(* Logix 5000 project; controller DUNEW2PLC1 vendor 1 type 14 code 221 rev 33.11; software revision 33.00; part 4 of 4 *)
(* tags used below, declared in another part *)
   ALL_EOT_GOOD : BOOL;
   HomeTrigger : BOOL;
   INIT_DONE : BOOL;
   MORE_STATS_S : BOOL[32];
   MOVE_TYPE : INT;   // 0 = No Move 1 = XY JOG 2 = XY Plane Move 3 = Z JOG 4 = Z Axis Move 5 = Toggle Latch Actuator 6 = Home the Latch Actuator
   NEXTSTATE : DINT;
   resetPB_S : BOOL;
   Safety_System_Healthy : BOOL;
   Safety_Tripped_S : BOOL;
   STATE : DINT;   // CURRENT State Machine State
   X_axis : AXIS_CIP_DRIVE;
   X_Axis_SFX : SAFETY_FEEDBACK_INTERFACE;
   X_Axis_SLS : SAFELY_LIMITED_SPEED;
   Y_axis : AXIS_CIP_DRIVE;
   Z_axis : AXIS_CIP_DRIVE;

PROGRAM Ready_State_1   (* main routine Ready *)
VAR
   OutBit : BOOL[32];
   SetBit : BOOL[32];
   STATE1_IND : BOOL := 1; {access Read Only}
END_VAR

ROUTINE Ready   (* ladder *)
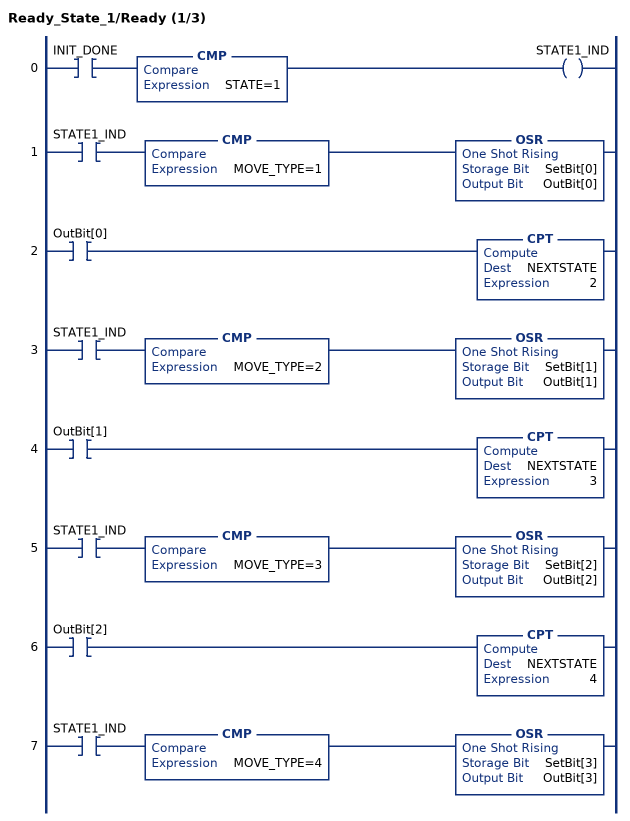
   0: XIC(INIT_DONE)CMP(STATE=1)OTE(STATE1_IND);
   1: XIC(STATE1_IND)CMP(MOVE_TYPE=1)OSR(SetBit[0],OutBit[0]);
   2: XIC(OutBit[0])CPT(NEXTSTATE,2);
   3: XIC(STATE1_IND)CMP(MOVE_TYPE=2)OSR(SetBit[1],OutBit[1]);
   4: XIC(OutBit[1])CPT(NEXTSTATE,3);
   5: XIC(STATE1_IND)CMP(MOVE_TYPE=3)OSR(SetBit[2],OutBit[2]);
   6: XIC(OutBit[2])CPT(NEXTSTATE,4);
   7: XIC(STATE1_IND)CMP(MOVE_TYPE=4)OSR(SetBit[3],OutBit[3]);
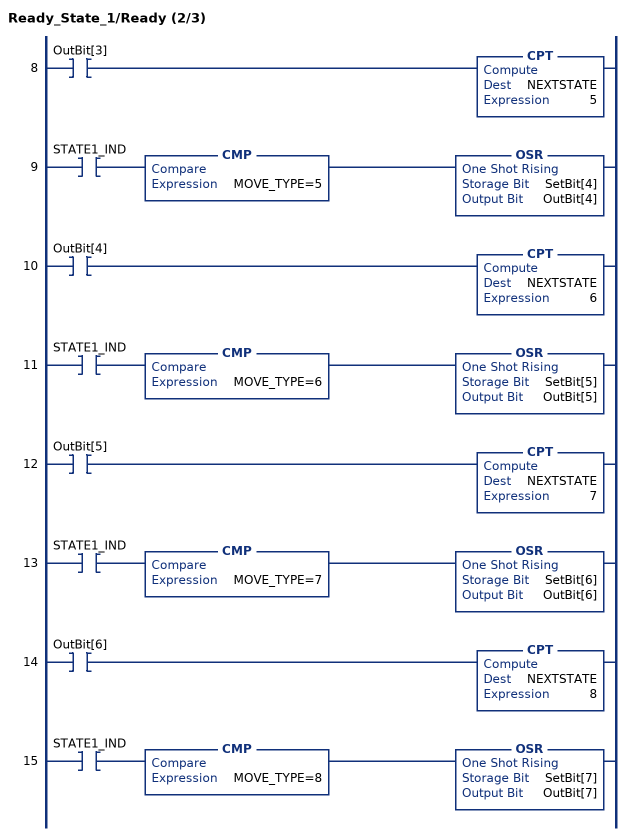
   8: XIC(OutBit[3])CPT(NEXTSTATE,5);
   9: XIC(STATE1_IND)CMP(MOVE_TYPE=5)OSR(SetBit[4],OutBit[4]);
   10: XIC(OutBit[4])CPT(NEXTSTATE,6);
   11: XIC(STATE1_IND)CMP(MOVE_TYPE=6)OSR(SetBit[5],OutBit[5]);
   12: XIC(OutBit[5])CPT(NEXTSTATE,7);
   13: XIC(STATE1_IND)CMP(MOVE_TYPE=7)OSR(SetBit[6],OutBit[6]);
   14: XIC(OutBit[6])CPT(NEXTSTATE,8);
   15: XIC(STATE1_IND)CMP(MOVE_TYPE=8)OSR(SetBit[7],OutBit[7]);
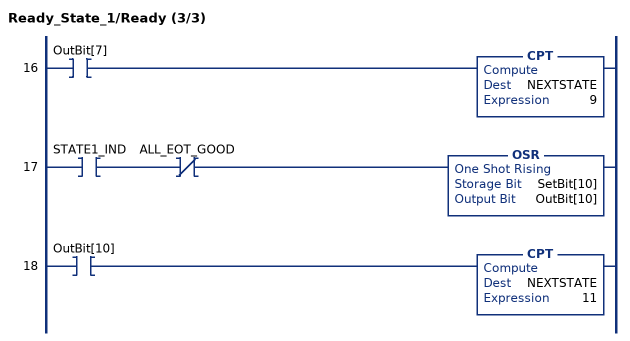
   16: XIC(OutBit[7])CPT(NEXTSTATE,9);
   17 (stored rung type 4): XIC(STATE1_IND)XIO(ALL_EOT_GOOD)OSR(SetBit[10],OutBit[10]);
   18 (stored rung type 4): XIC(OutBit[10])CPT(NEXTSTATE,11);
END_ROUTINE
END_PROGRAM

PROGRAM Safety   (* main routine Safety, safety *)
VAR
   e : BOOL;
   Machine_Reduced_Speed : BOOL;
END_VAR

ROUTINE Safety   (* ladder *)
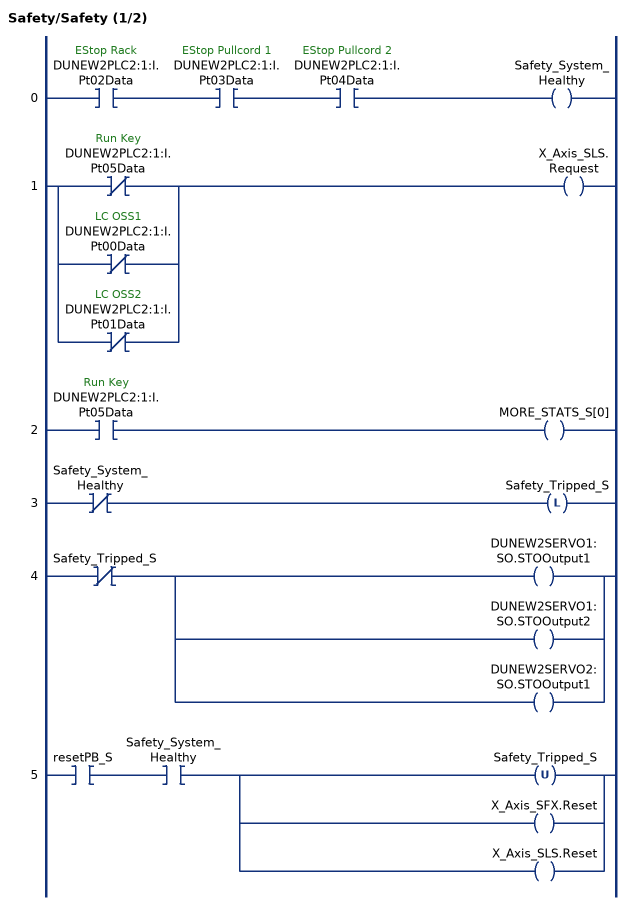
   0: XIC(DUNEW2PLC2:1:I.Pt02Data)XIC(DUNEW2PLC2:1:I.Pt03Data)XIC(DUNEW2PLC2:1:I.Pt04Data)OTE(Safety_System_Healthy);
   1: [XIO(DUNEW2PLC2:1:I.Pt05Data) ,XIO(DUNEW2PLC2:1:I.Pt00Data) ,XIO(DUNEW2PLC2:1:I.Pt01Data) ]OTE(X_Axis_SLS.Request);
   2: XIC(DUNEW2PLC2:1:I.Pt05Data)OTE(MORE_STATS_S[0]);
   3: XIO(Safety_System_Healthy)OTL(Safety_Tripped_S);
   4: XIO(Safety_Tripped_S)[[OTE(DUNEW2SERVO1:SO.STOOutput1) ,OTE(DUNEW2SERVO1:SO.STOOutput2) ] ,OTE(DUNEW2SERVO2:SO.STOOutput1) ];
   5: XIC(resetPB_S)XIC(Safety_System_Healthy)[OTU(Safety_Tripped_S) ,[OTE(X_Axis_SFX.Reset) ,OTE(X_Axis_SLS.Reset) ] ];
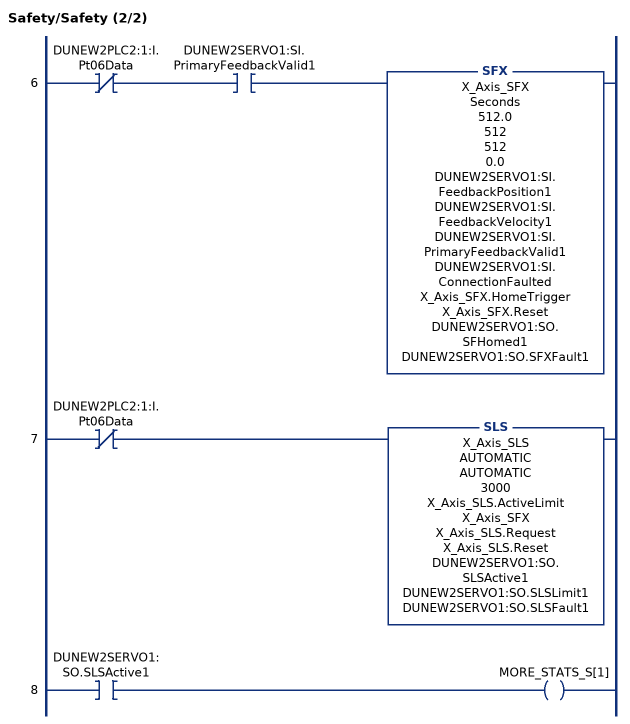
   6: XIO(DUNEW2PLC2:1:I.Pt06Data)XIC(DUNEW2SERVO1:SI.PrimaryFeedbackValid1)SFX(X_Axis_SFX,Seconds,512.0,512,512,0.0,DUNEW2SERVO1:SI.FeedbackPosition1,DUNEW2SERVO1:SI.FeedbackVelocity1,DUNEW2SERVO1:SI.PrimaryFeedbackValid1,DUNEW2SERVO1:SI.ConnectionFaulted,X_Axis_SFX.HomeTrigger,X_Axis_SFX.Reset,DUNEW2SERVO1:SO.SFHomed1,DUNEW2SERVO1:SO.SFXFault1);
   7: XIO(DUNEW2PLC2:1:I.Pt06Data)SLS(X_Axis_SLS,AUTOMATIC,AUTOMATIC,3000,X_Axis_SLS.ActiveLimit,X_Axis_SFX,X_Axis_SLS.Request,X_Axis_SLS.Reset,DUNEW2SERVO1:SO.SLSActive1,DUNEW2SERVO1:SO.SLSLimit1,DUNEW2SERVO1:SO.SLSFault1);
   8: XIC(DUNEW2SERVO1:SO.SLSActive1)OTE(MORE_STATS_S[1]);
END_ROUTINE
END_PROGRAM

PROGRAM UnServo_9   (* main routine UnServo_All *)
VAR
   oneshotob : BOOL[32]; {access Read Only}
   oneshotsb : BOOL[32]; {access Read Only}
   STATE9_IND : BOOL; {access Read Only}
   X_AXIS_STAT : MOTION_INSTRUCTION[32] := ([0].FLAGS := 33554432, [1].FLAGS := 33554432, [2].FLAGS := 536870912, [2].DN := 1, [2].STATE := 1); {access Read Only}
   Y_AXIS_STAT : MOTION_INSTRUCTION[32] := ([0].FLAGS := 33554432, [1].FLAGS := 33554432, [2].FLAGS := 536870912, [2].DN := 1, [2].STATE := 1); {access Read Only}
   Z_AXIS_STAT : MOTION_INSTRUCTION[32] := ([0].FLAGS := 33554432, [1].FLAGS := 33554432, [2].FLAGS := 536870912, [2].DN := 1, [2].STATE := 1); {access Read Only}
END_VAR

ROUTINE UnServo_All   (* ladder *)
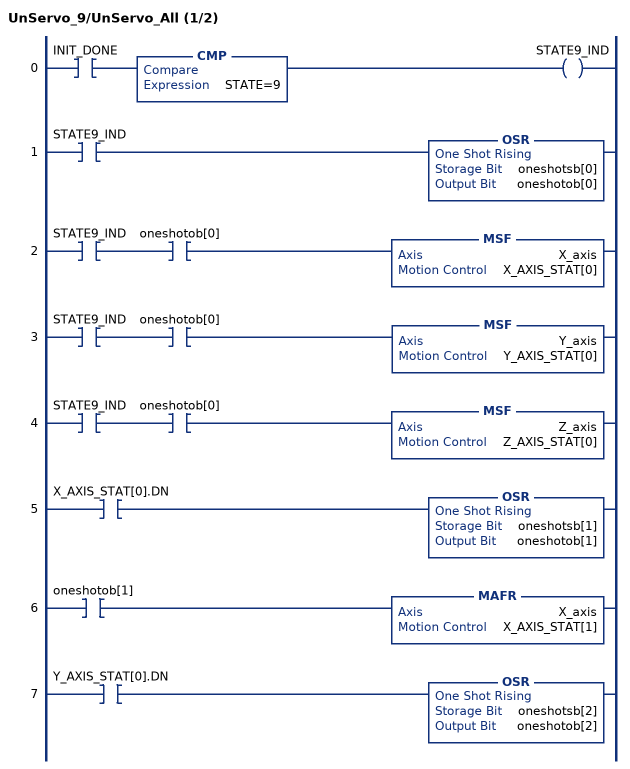
   0: XIC(INIT_DONE)CMP(STATE=9)OTE(STATE9_IND);
   1: XIC(STATE9_IND)OSR(oneshotsb[0],oneshotob[0]);
   2: XIC(STATE9_IND)XIC(oneshotob[0])MSF(X_axis,X_AXIS_STAT[0]);
   3: XIC(STATE9_IND)XIC(oneshotob[0])MSF(Y_axis,Y_AXIS_STAT[0]);
   4: XIC(STATE9_IND)XIC(oneshotob[0])MSF(Z_axis,Z_AXIS_STAT[0]);
   5: XIC(X_AXIS_STAT[0].DN)OSR(oneshotsb[1],oneshotob[1]);
   6: XIC(oneshotob[1])MAFR(X_axis,X_AXIS_STAT[1]);
   7: XIC(Y_AXIS_STAT[0].DN)OSR(oneshotsb[2],oneshotob[2]);
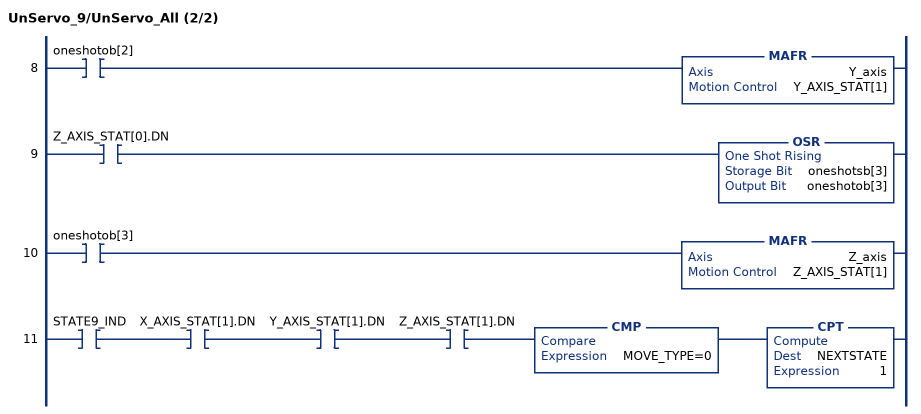
   8: XIC(oneshotob[2])MAFR(Y_axis,Y_AXIS_STAT[1]);
   9: XIC(Z_AXIS_STAT[0].DN)OSR(oneshotsb[3],oneshotob[3]);
   10: XIC(oneshotob[3])MAFR(Z_axis,Z_AXIS_STAT[1]);
   11: XIC(STATE9_IND)XIC(X_AXIS_STAT[1].DN)XIC(Y_AXIS_STAT[1].DN)XIC(Z_AXIS_STAT[1].DN)CMP(MOVE_TYPE=0)CPT(NEXTSTATE,1);
END_ROUTINE
END_PROGRAM
